{attribute addProperty BoxType "EK1100-0000-0018"}
{attribute addProperty Id "Beckhoff_EJ3xxxEK1122Beckhoff_EJ3xxxEK1122_6922078E162A_0001_EJ3004_0000_0019EJ3004_360D511E40650.75A_0002_EJ3004_0000_0020EJ3004_19668D2840650.75A_0003_EJ3004_0000_0021EJ3004_19668D2840650.75A_0004_EJ3048_0000_0020EJ3048_EA60A07733842.25A_0005_EJ3058_0000_0020EJ3058_EA60A07733842.25A_0006_EJ3068_0000_0020EJ3068_EA60A07733842.25A_0007_EJ3068_0000_0021EJ3068_EA60A07733842.25A_0008_EJ3104_0000_0019EJ3104_B7B5302521026.25A_0009_EJ3104_0000_0020EJ3104_B7B5302521026.25A_0010_EJ3104_0000_0021EJ3104_B7B5302521026.25A_0011_EJ3108_0000_0017EJ3108_EA60A07733842.25A_0012_EJ3108_0000_0018EJ3108_060F55FF33842.25A_0013_EJ3108_0000_0019EJ3108_060F55FF33842.25A_0014_EJ3202_0000_0019EJ3202_CEE8F25A24430.5A_0015_EJ3202_0000_0020EJ3202_CEE8F25A24430.5A_0016_EJ3202_0000_0021EJ3202_CEE8F25A24430.5A_0017_EJ3214_0000_0016EJ3214_712ECA1B21026.25A_0018_EJ3255_0000_0023EJ3255_7B3AD95824230.25A_0019_EJ3318_0000_0017EJ3318_4B9E477A40250.25"}
{attribute addProperty CRC "3770829976"}
{attribute addProperty SizeInBites "5816"}
{attribute addProperty SizeInBytes "727"}
TYPE Beckhoff_EJ3xxx_E0C24C98 EXTENDS EK1100_179A0949 :
STRUCT
	{attribute addProperty Name "Beckhoff_EJ3xxxEK1122"}
	Beckhoff_EJ3xxxEK1122 : Beckhoff_EJ3xxxEK1122_6922078E;
	{attribute addProperty Name "A_0001_EJ3004_0000_0019"}
	A_0001_EJ3004_0000_0019 : EJ3004_360D511E;
	{attribute addProperty Name "A_0002_EJ3004_0000_0020"}
	A_0002_EJ3004_0000_0020 : EJ3004_19668D28;
	{attribute addProperty Name "A_0003_EJ3004_0000_0021"}
	A_0003_EJ3004_0000_0021 : EJ3004_19668D28;
	{attribute addProperty Name "A_0004_EJ3048_0000_0020"}
	A_0004_EJ3048_0000_0020 : EJ3048_EA60A077;
	{attribute addProperty Name "A_0005_EJ3058_0000_0020"}
	A_0005_EJ3058_0000_0020 : EJ3058_EA60A077;
	{attribute addProperty Name "A_0006_EJ3068_0000_0020"}
	A_0006_EJ3068_0000_0020 : EJ3068_EA60A077;
	{attribute addProperty Name "A_0007_EJ3068_0000_0021"}
	A_0007_EJ3068_0000_0021 : EJ3068_EA60A077;
	{attribute addProperty Name "A_0008_EJ3104_0000_0019"}
	A_0008_EJ3104_0000_0019 : EJ3104_B7B53025;
	{attribute addProperty Name "A_0009_EJ3104_0000_0020"}
	A_0009_EJ3104_0000_0020 : EJ3104_B7B53025;
	{attribute addProperty Name "A_0010_EJ3104_0000_0021"}
	A_0010_EJ3104_0000_0021 : EJ3104_B7B53025;
	{attribute addProperty Name "A_0011_EJ3108_0000_0017"}
	A_0011_EJ3108_0000_0017 : EJ3108_EA60A077;
	{attribute addProperty Name "A_0012_EJ3108_0000_0018"}
	A_0012_EJ3108_0000_0018 : EJ3108_060F55FF;
	{attribute addProperty Name "A_0013_EJ3108_0000_0019"}
	A_0013_EJ3108_0000_0019 : EJ3108_060F55FF;
	{attribute addProperty Name "A_0014_EJ3202_0000_0019"}
	A_0014_EJ3202_0000_0019 : EJ3202_CEE8F25A;
	{attribute addProperty Name "A_0015_EJ3202_0000_0020"}
	A_0015_EJ3202_0000_0020 : EJ3202_CEE8F25A;
	{attribute addProperty Name "A_0016_EJ3202_0000_0021"}
	A_0016_EJ3202_0000_0021 : EJ3202_CEE8F25A;
	{attribute addProperty Name "A_0017_EJ3214_0000_0016"}
	A_0017_EJ3214_0000_0016 : EJ3214_712ECA1B;
	{attribute addProperty Name "A_0018_EJ3255_0000_0023"}
	A_0018_EJ3255_0000_0023 : EJ3255_7B3AD958;
	{attribute addProperty Name "A_0019_EJ3318_0000_0017"}
	A_0019_EJ3318_0000_0017 : EJ3318_4B9E477A;
END_STRUCT
END_TYPE

(* stored: Version 1.2.0.0, ProductVersion 3.1.4024.9
   DUT Beckhoff_EJ3xxx_E0C24C98: Id {4015f189-57cb-4495-b16f-dc632d15db8d} *)
